FUNCTION_BLOCK FB_PackML_PushButtonControl EXTENDS FB_PackML_ExternalControl
VAR_INPUT
END_VAR
VAR_OUTPUT
END_VAR
VAR
	bStartButton	AT %I* : BOOL;	//Tie to hardware start pushbutton
	//TODO: add other buttons
END_VAR

//TODO: implement button control

END_FUNCTION_BLOCK

(* stored: Version 1.1.0.1, ProductVersion 3.1.4024.10
   POU FB_PackML_PushButtonControl: Id {6be5865f-6c78-4181-b3c0-db233d854256}, SpecialFunc None *)
